FUNCTION PressureToFlow : LREAL
VAR_INPUT
	Pressure: LREAL;
	k: LREAL;
END_VAR
VAR
	DiffPressure: LREAL;
END_VAR

DiffPressure := Pressure;
IF diffpressure < 0 THEN
	DiffPressure := 0;
END_IF 
PressureToFlow := k * SQRT(DiffPressure);// / 3.6;

END_FUNCTION

(* stored: Version 1.1.0.1, ProductVersion 3.1.4024.6
   POU PressureToFlow: Id {cd526757-80b0-4a2d-a96c-969d2b1d009d}, SpecialFunc None *)
